// SIMATIC S7-200 project (STEP 7-Micro/WIN), CPU 224XP REL 02.01

SYMBOL_TABLE USUARIO1
UP               I0.0     // UP INCREMENTO EN UNA UNIDAD
DOWN             I0.1     // DOWN DECREMENTO EN UNA UNIDAD
RESET            I0.2     // RESET PUESTA A CERO DE LA CUENTA
CONTADOR1        MW0      // CONTADOR DEL PROGRAMA
DISPLAY1         MB2      // PARA MOSTRAR EL VALOR DE LA CUENTA EN D1
DISPLAY2         MB3      // PARA MOSTRAR EL VALOR DE LA CUENTA EN D2
CONTADOR2        MW4      // CONTADOR DE LAS DECENAS
END_SYMBOL_TABLE

ORGANIZATION_BLOCK PRINCIPAL:OB1
TITLE=COMENTARIOS DEL PROGRAMA
BEGIN
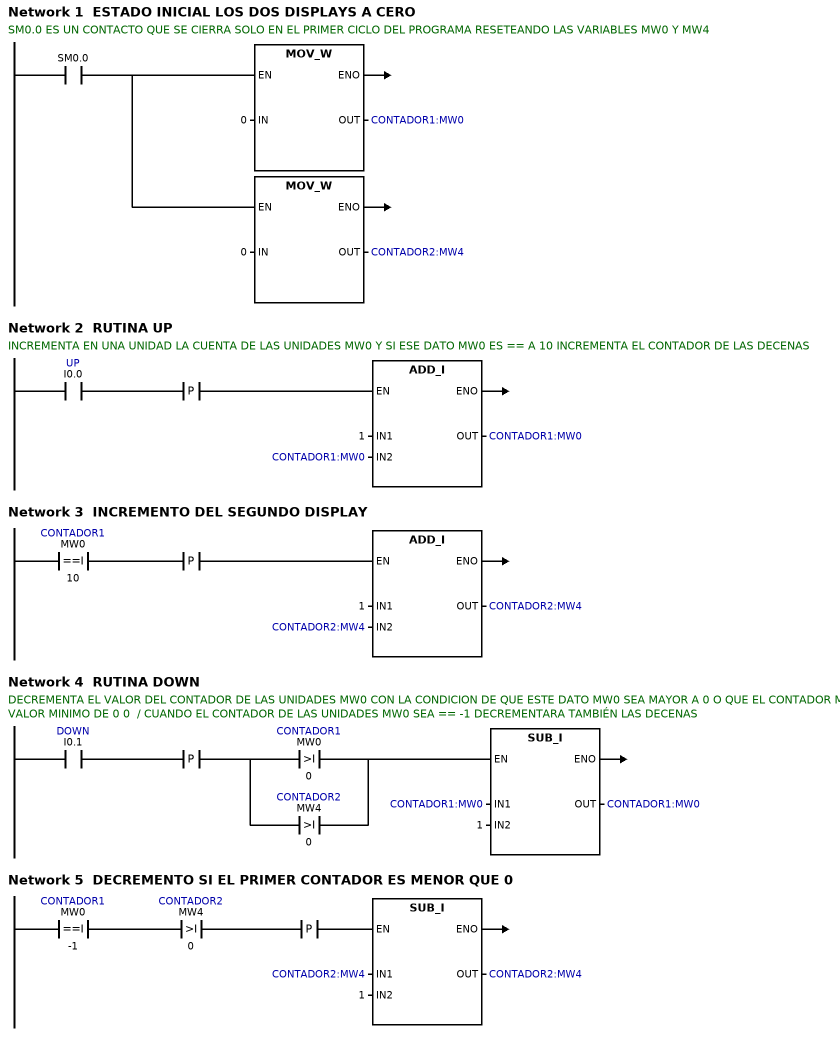
Network 1 // ESTADO INICIAL LOS DOS DISPLAYS A CERO
// SM0.0 ES UN CONTACTO QUE SE CIERRA SOLO EN EL PRIMER CICLO DEL PROGRAMA RESETEANDO LAS VARIABLES MW0 Y MW4
LD     SM0.0
MOVW   0, CONTADOR1:MW0
MOVW   0, CONTADOR2:MW4
Network 2 // RUTINA UP
// INCREMENTA EN UNA UNIDAD LA CUENTA DE LAS UNIDADES MW0 Y SI ESE DATO MW0 ES == A 10 INCREMENTA EL CONTADOR DE LAS DECENAS
// (network saved uncompiled; LAD cells follow)
// row 0: c0 -| |- UP:I0.0  c1 -|P|-  c2 --  c3 [ADD_I EN:=power@row0, IN1:=1, IN2:=CONTADOR1:MW0, ENO=>power, OUT=>CONTADOR1:MW0]  c4 ->
// row 1: c3 [box]
Network 3 // INCREMENTO DEL SEGUNDO DISPLAY
// (network saved uncompiled; LAD cells follow)
// row 0: c0 -|==I|- CONTADOR1:MW0, 10  c1 -|P|-  c2 --  c3 [ADD_I EN:=power@row0, IN1:=1, IN2:=CONTADOR2:MW4, ENO=>power, OUT=>CONTADOR2:MW4]  c4 ->
// row 1: c3 [box]
Network 4 // RUTINA DOWN	
// DECREMENTA EL VALOR DEL CONTADOR DE LAS UNIDADES MW0 CON LA CONDICION DE QUE ESTE DATO MW0 SEA MAYOR A 0 O QUE EL CONTADOR MW4 SEA MAYOR QUE 0 PARA QUE LLEGUE AL VALOR MINIMO DE 0 0 
// CUANDO EL CONTADOR DE LAS UNIDADES MW0 SEA == -1 DECREMENTARA TAMBIÉN LAS DECENAS
// (network saved uncompiled; LAD cells follow)
// row 0: c0 -| |- DOWN:I0.1  c1 -|P|-  v  c2 -|>I|- CONTADOR1:MW0, 0 v  c3 --  c4 [SUB_I EN:=power@row0, IN1:=CONTADOR1:MW0, IN2:=1, ENO=>power, OUT=>CONTADOR1:MW0]  c5 ->
// row 1: c1 ^  c2 -|>I|- CONTADOR2:MW4, 0 ^  c4 [box]
Network 5 // DECREMENTO SI EL PRIMER CONTADOR ES MENOR QUE 0
// (network saved uncompiled; LAD cells follow)
// row 0: c0 -|==I|- CONTADOR1:MW0, -1  c1 -|>I|- CONTADOR2:MW4, 0  c2 -|P|-  c3 [SUB_I EN:=power@row0, IN1:=CONTADOR2:MW4, IN2:=1, ENO=>power, OUT=>CONTADOR2:MW4]  c4 ->
// row 1: c3 [box]
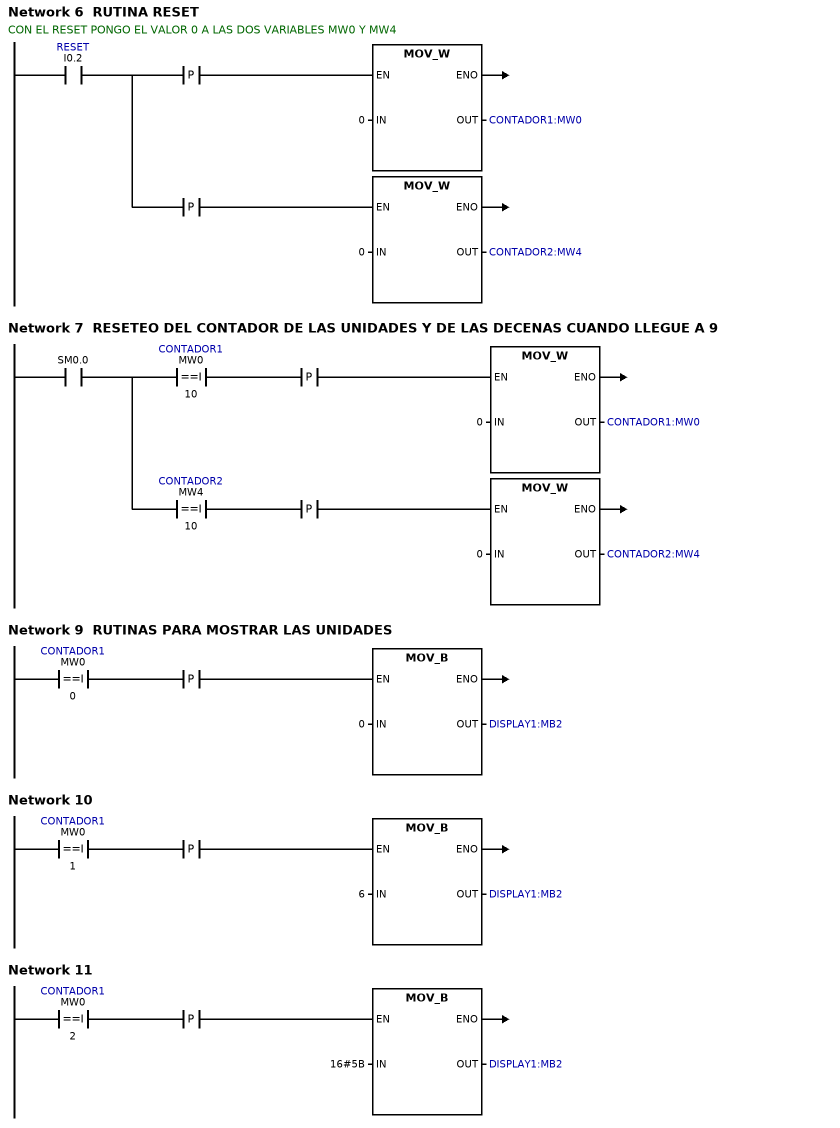
Network 6 // RUTINA RESET
// CON EL RESET PONGO EL VALOR 0 A LAS DOS VARIABLES MW0 Y MW4
LD     RESET:I0.2
LPS
EU
MOVW   0, CONTADOR1:MW0
LPP
EU
MOVW   0, CONTADOR2:MW4
Network 7 // RESETEO DEL CONTADOR DE LAS UNIDADES Y DE LAS DECENAS CUANDO LLEGUE A 9
LD     SM0.0
LPS
AW=    CONTADOR1:MW0, 10
EU
MOVW   0, CONTADOR1:MW0
LPP
AW=    CONTADOR2:MW4, 10
EU
MOVW   0, CONTADOR2:MW4
Network 9 // RUTINAS PARA MOSTRAR LAS UNIDADES
LDW=   CONTADOR1:MW0, 0
EU
MOVB   0, DISPLAY1:MB2
Network 10
LDW=   CONTADOR1:MW0, 1
EU
MOVB   6, DISPLAY1:MB2
Network 11
LDW=   CONTADOR1:MW0, 2
EU
MOVB   16#5B, DISPLAY1:MB2
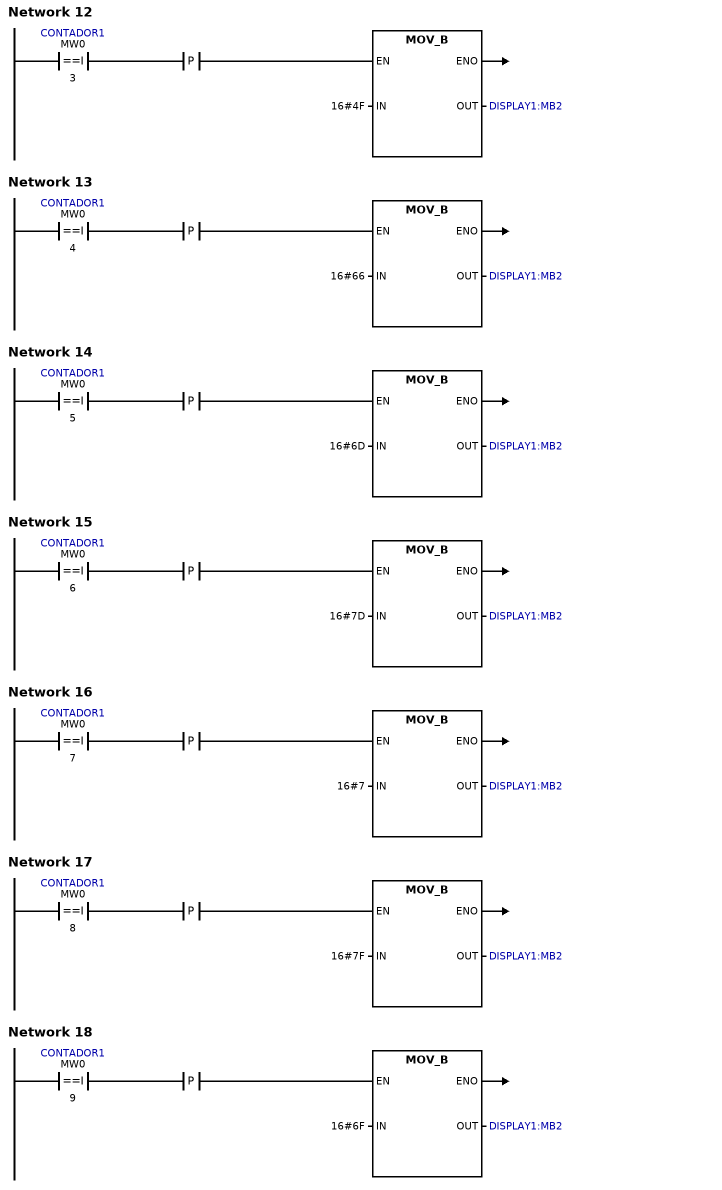
Network 12
LDW=   CONTADOR1:MW0, 3
EU
MOVB   16#4F, DISPLAY1:MB2
Network 13
LDW=   CONTADOR1:MW0, 4
EU
MOVB   16#66, DISPLAY1:MB2
Network 14
LDW=   CONTADOR1:MW0, 5
EU
MOVB   16#6D, DISPLAY1:MB2
Network 15
LDW=   CONTADOR1:MW0, 6
EU
MOVB   16#7D, DISPLAY1:MB2
Network 16
LDW=   CONTADOR1:MW0, 7
EU
MOVB   16#7, DISPLAY1:MB2
Network 17
LDW=   CONTADOR1:MW0, 8
EU
MOVB   16#7F, DISPLAY1:MB2
Network 18
LDW=   CONTADOR1:MW0, 9
EU
MOVB   16#6F, DISPLAY1:MB2
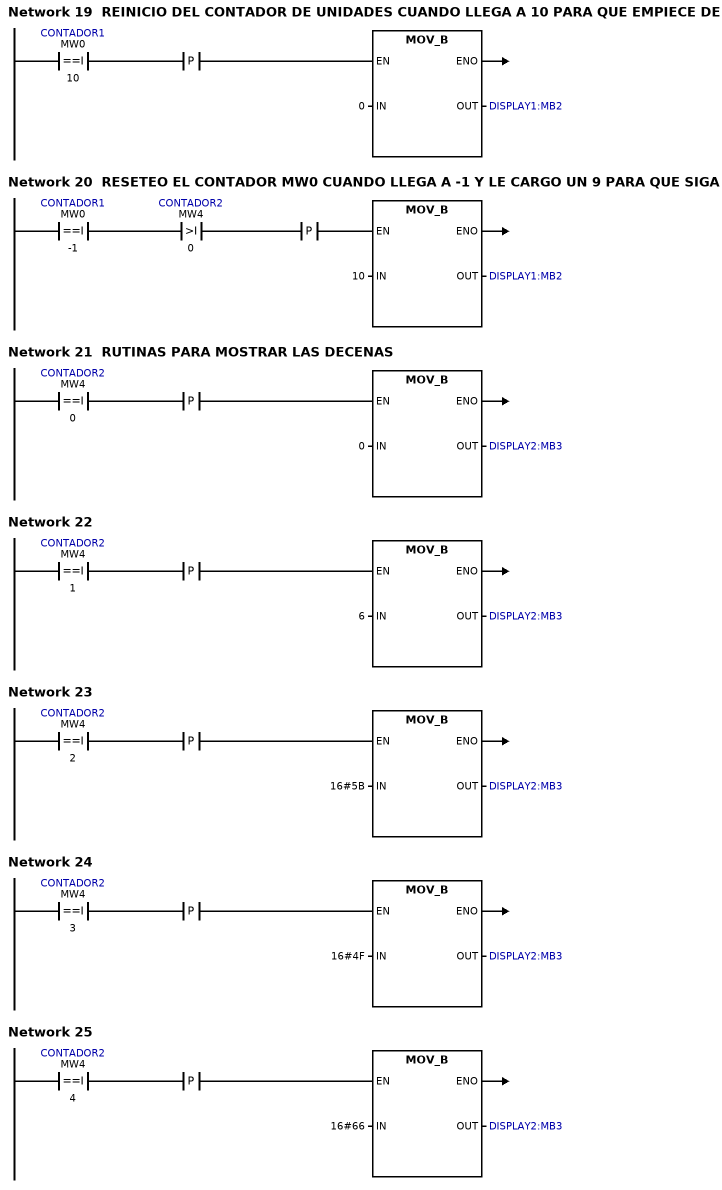
Network 19 // REINICIO DEL CONTADOR DE UNIDADES CUANDO LLEGA A 10 PARA QUE EMPIECE DE NUEVO EN 0
LDW=   CONTADOR1:MW0, 10
EU
MOVB   0, DISPLAY1:MB2
Network 20 // RESETEO EL CONTADOR MW0 CUANDO LLEGA A -1 Y LE CARGO UN 9 PARA QUE SIGA DECREMENTANDO
// (network saved uncompiled; LAD cells follow)
// row 0: c0 -|==I|- CONTADOR1:MW0, -1  c1 -|>I|- CONTADOR2:MW4, 0  c2 -|P|-  c3 [MOV_B EN:=power@row0, IN:=10, ENO=>power, OUT=>DISPLAY1:MB2]  c4 ->
// row 1: c3 [box]
Network 21 // RUTINAS PARA MOSTRAR LAS DECENAS
LDW=   CONTADOR2:MW4, 0
EU
MOVB   0, DISPLAY2:MB3
Network 22
LDW=   CONTADOR2:MW4, 1
EU
MOVB   6, DISPLAY2:MB3
Network 23
LDW=   CONTADOR2:MW4, 2
EU
MOVB   16#5B, DISPLAY2:MB3
Network 24
LDW=   CONTADOR2:MW4, 3
EU
MOVB   16#4F, DISPLAY2:MB3
Network 25
LDW=   CONTADOR2:MW4, 4
EU
MOVB   16#66, DISPLAY2:MB3
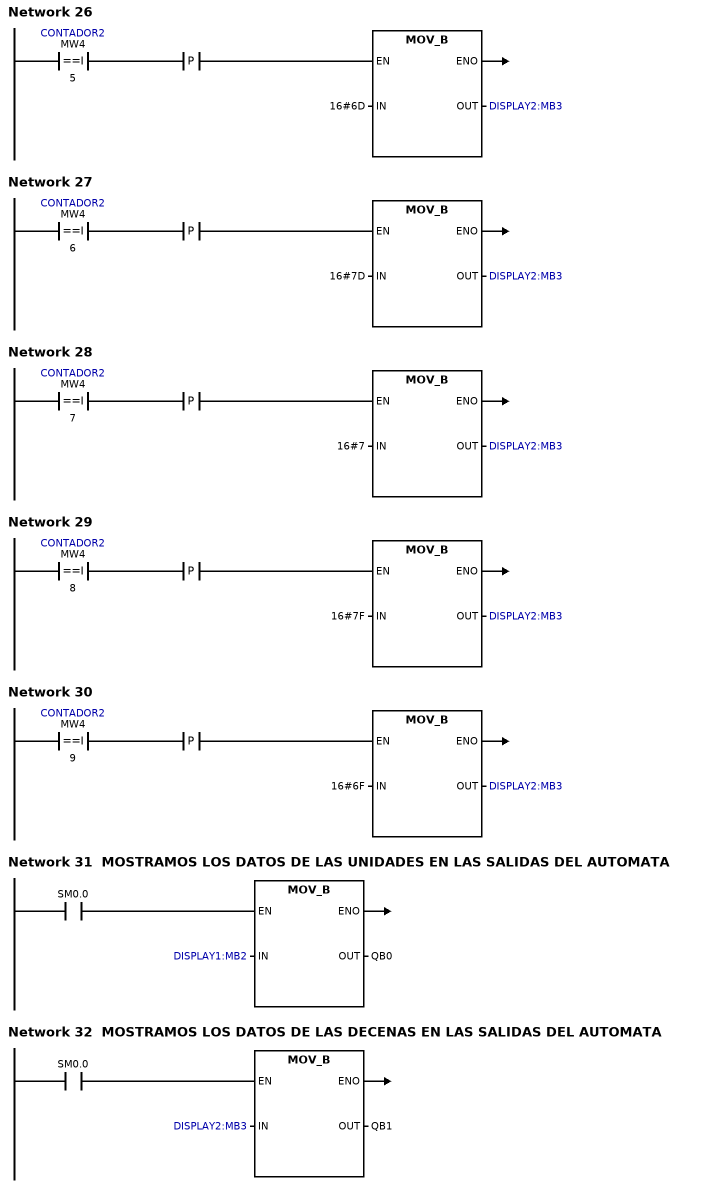
Network 26
LDW=   CONTADOR2:MW4, 5
EU
MOVB   16#6D, DISPLAY2:MB3
Network 27
LDW=   CONTADOR2:MW4, 6
EU
MOVB   16#7D, DISPLAY2:MB3
Network 28
LDW=   CONTADOR2:MW4, 7
EU
MOVB   16#7, DISPLAY2:MB3
Network 29
LDW=   CONTADOR2:MW4, 8
EU
MOVB   16#7F, DISPLAY2:MB3
Network 30
LDW=   CONTADOR2:MW4, 9
EU
MOVB   16#6F, DISPLAY2:MB3
Network 31 // MOSTRAMOS LOS DATOS DE LAS UNIDADES EN LAS SALIDAS DEL AUTOMATA
LD     SM0.0
MOVB   DISPLAY1:MB2, QB0
Network 32 // MOSTRAMOS LOS DATOS DE LAS DECENAS EN LAS SALIDAS DEL AUTOMATA
LD     SM0.0
MOVB   DISPLAY2:MB3, QB1
END_ORGANIZATION_BLOCK
